Fanuc KAREL source: kb00135.KL

-- PROVISIONAL review KL for V770-1; original PC SHA256 9047b6f9a6bb65160f1171d097644c089059ef7cd540f8ad6f225bfdce7e98ad
-- Incomplete behavior may be omitted. Consult companion uncertainty JSON. Do not deploy.
PROGRAM KB00135
%NOLOCKGROUP
BEGIN
  -- UNRESOLVED_PC offsets 5-12; opcodes 9D,23
  -- UNRESOLVED_PC offsets 17-26; opcodes 3F,75
  -- UNRESOLVED_PC offsets 31-38; opcodes 9D,23
  -- UNRESOLVED_PC offsets 43-50; opcodes 9D,23
  -- UNRESOLVED_PC offsets 55-85; opcodes 27,22,22,2A,22,22,31
  -- UNRESOLVED_PC offsets 90-94; opcodes 7F
END KB00135
